// TwinCAT 3 PLC project Untitled1
// ProgramVersion: 3.1.4023.0
// libraries:
//   Tc2_MC2, * (Beckhoff Automation GmbH)
//   Tc2_Standard, * (Beckhoff Automation GmbH)
//   Tc2_System, * (Beckhoff Automation GmbH)
//   Tc2_Utilities, * (Beckhoff Automation GmbH)
//   Tc3_JsonXml, * (Beckhoff Automation GmbH)
//   Tc3_Module, * (Beckhoff Automation GmbH)
//   Tc3_PackML_V2, * (Beckhoff Automation GmbH)
// project tree:
//   DUTs/ Bundle.TcDUT (not stored), Interval.TcDUT (not stored), PositionMaterials.TcDUT (not stored)
//   DUTs/Enums/ TaskA22.TcDUT (not stored), Cardboard.TcDUT (not stored), CornerGuard.TcDUT (not stored), E_PMLCustomUnitMode.TcDUT (not stored), SectionEnum.TcDUT (not stored), Surface.TcDUT (not stored)
//   DUTs/Insertion Package/Drives/ AirPiston.TcPOU (not stored), ClearLinkMC.TcPOU (not stored), ServoNC.TcPOU (not stored), SimplePiston.TcPOU (not stored)
//   DUTs/Insertion Package/ Homing.TcDUT (not stored), Insertion.TcPOU (not stored), SuctionPad.TcDUT (not stored)
//   DUTs/Insertion Package/Prototypes/ FBA_Drive.TcPOU (not stored), FBA_TrifectaDrive.TcPOU (not stored), I_ContinuousDrive.TcIO (not stored), I_Drive.TcIO (not stored), I_EncodedDrive.TcIO (not stored), I_PositionalDrive.TcIO (not stored)
//   DUTs/Machines/ FoldingMachine.TcPOU, KukaRobot.TcPOU (not stored), RobotA22.TcPOU, WrapMachine.TcPOU
//   DUTs/Material Holders/ MaterialHolder.TcPOU (not stored), MaterialSlot.TcDUT (not stored), SkidMagazine.TcPOU (not stored)
//   GVLs/ ContainerArrays.TcGVL, GVL.TcGVL (not stored), Hardware.TcGVL, Misc.TcGVL (not stored)
//   / PlcTask.TcTTO (not stored)
//   POUs/A22 - Cardboard + Guard/AOIs/ AOI_LoadCornerCardboard.TcPOU (not stored), AOI_LoadCornerGuard.TcPOU, AOI_LoadFlatCardboard.TcPOU
//   POUs/A22 - Cardboard + Guard/ FiberboardEx.TcPOU
//   POUs/ FB_System.TcPOU (not stored), MAIN.TcPOU, BundleToJson.TcPOU (not stored)
//   POUs/Hardware Calls/ SuctionQualityPtr.TcPOU (not stored), SetSuctionsPtrArr.TcPOU (not stored), CallHardwareModules.TcPOU, SuctionQuality.TcPOU (not stored), SetSuctions.TcPOU (not stored), SetupHardware.TcPOU (not stored)
//   POUs/Materials/ GetMaterialLength.TcPOU (not stored), GetMaterialLengthFromCode.TcPOU (not stored), GetPairMasterLength.TcPOU (not stored), GetPositionMasterLength.TcPOU (not stored), MatchesMaterialType.TcPOU (not stored)
//   POUs/Utility/ CEILING.TcPOU (not stored), IntegerBitAccess.TcPOU (not stored), IntegerToBoolArray.TcPOU (not stored), WithinTolerance.TcPOU (not stored)
// real-time tasks:
//   TASK PlcTask: cycle T#10ms, priority 20, ADS port 350
// motion (NC):
//   TASK NC-Task 1 SAF: cycle T#2ms, priority 4, ADS port 501
//   TASK NC-Task 1 SVB: cycle T#10ms, priority 8, ADS port 511
//   AXIS A22_IM_HS_L (id 1)
//     OtherSettings: AllowMotionCmdToSlave=true
//     encoder EncType=19
//       EncPara: MaxCount=#xffffffff
//     drive DrvType=16
//       DrvPara: MaxCount=#xffffffff
//         Analog: TorqueSetpointScale=10, ScaleFactorActTorque=0.1
//         TimeComp: TaskDelayCycles=1
//     controller CtrType=1
//       CtrPara: PriorControlFactor=1
//         Observer: BandWidth=20
//   AXIS A22_IM_HS_R (id 2)
//     OtherSettings: AllowMotionCmdToSlave=true
//     encoder EncType=19
//       EncPara: MaxCount=#xffffffff
//     drive DrvType=16
//       DrvPara: MaxCount=#xffffffff, DriveControlDWord=#x00000100
//         Analog: TorqueSetpointScale=10, ScaleFactorActTorque=0.1
//         TimeComp: TaskDelayCycles=1
//     controller CtrType=1
//       CtrPara: PriorControlFactor=1
//         Observer: BandWidth=20
// I/O:
//   DEVICE Device 1 (EtherCAT) (disabled), AmsNetId 192.168.101.188.2.1
//     EK1200 [EK1200-5000 EtherCAT Power supply (2A E-Bus)]
//       IPC_O [EL2809 16Ch. Dig. Output 24V, 0.5A]
//       JUNC_1 [EK1122 2 port EtherCAT junction]
//         A21_C4 [EK1100 EtherCAT Coupler (2A E-Bus)]
//           A21_C4_I1 [EL1809 16Ch. Dig. Input 24V, 3ms]
//           A21_C4_O2 [EL2809 16Ch. Dig. Output 24V, 0.5A]
//           A21_C4_O3 [EL2809 16Ch. Dig. Output 24V, 0.5A]
//           BRIDGE_ROBOT1 [EL6695 EtherCAT Bridge terminal (Primary)]
//           A21_C4_END [EL9011 End Terminal]
//         A21_SB01 [EP1809-0021 16 Ch. Dig. Input 24V, 3ms, M8]
//         A21_SB05 [EP1008-0001 8 Ch. Dig. Input 24V, 3ms, M8]
//         A21_SB04 [EP1809-0021 16 Ch. Dig. Input 24V, 3ms, M8]
//         A21_SB03 [EP1008-0001 8 Ch. Dig. Input 24V, 3ms, M8]
//         A21_C1 [EK1100 EtherCAT Coupler (2A E-Bus)]
//           A21_C1_I1 [EL1809 16Ch. Dig. Input 24V, 3ms]
//           A21_C1_O2 [EL2809 16Ch. Dig. Output 24V, 0.5A]
//           BRIDGE_ROBOT2 [EL6695 EtherCAT Bridge terminal (Primary)]
//           A21_C1_END [EL9011 End Terminal]
//         A21_SB02 [EP1809-0021 16 Ch. Dig. Input 24V, 3ms, M8]
//         A21_SB07 [EP1008-0001 8 Ch. Dig. Input 24V, 3ms, M8]
//         A21_SB06 [EP1008-0001 8 Ch. Dig. Input 24V, 3ms, M8]
//       JUNC_2 [EK1122 2 port EtherCAT junction]
//         A22_C1 [EK1100 EtherCAT Coupler (2A E-Bus)]
//           A22_C1_I1 [EL1809 16Ch. Dig. Input 24V, 3ms]
//           A22_C1_O2 [EL2809 16Ch. Dig. Output 24V, 0.5A]
//           A22_C1_JUNC [EK1122 2 port EtherCAT junction]
//             A22_C4 [EK1100 EtherCAT Coupler (2A E-Bus)]
//               A22_C4_I1 [EL1809 16Ch. Dig. Input 24V, 3ms]
//               A22_C4_O2 [EL2809 16Ch. Dig. Output 24V, 0.5A]
//               A22_C4_O3 [EL2809 16Ch. Dig. Output 24V, 0.5A]
//               Term 31 (EL9011) [EL9011 End Terminal]
//             A22_C4_NC2 [CD02 EtherCAT Drive (CoE)]
//             A22_C4_NC1_TEMP [EK1100 EtherCAT Coupler (2A E-Bus)]
//               Term 34 (EL1008) [EL1008 8Ch. Dig. Input 24V, 3ms]
//               Term 35 (EL2008) [EL2008 8Ch. Dig. Output 24V, 0.5A]
//               Term 36 (EL9011) [EL9011 End Terminal]
//             A22_SB01 [EP1809-0021 16 Ch. Dig. Input 24V, 3ms, M8]
//             A22_SB04 [EP1809-0021 16 Ch. Dig. Input 24V, 3ms, M8]
//             A22_SB05 [EP1008-0001 8 Ch. Dig. Input 24V, 3ms, M8]
//             A22_C5 [EK1100 EtherCAT Coupler (2A E-Bus)]
//               A22_C5_I1 [EL1809 16Ch. Dig. Input 24V, 3ms]
//               A22_C5_O2 [EL2809 16Ch. Dig. Output 24V, 0.5A]
//               A22_C5_END [EL9011 End Terminal]
//             A22_SB06 [EP1008-0001 8 Ch. Dig. Input 24V, 3ms, M8]
//             A22_C6 [EK1100 EtherCAT Coupler (2A E-Bus)]
//               A22_C6_I1 [EL1809 16Ch. Dig. Input 24V, 3ms]
//               A22_C6_O2 [EL2809 16Ch. Dig. Output 24V, 0.5A]
//               A22_C6_O3 [EL2809 16Ch. Dig. Output 24V, 0.5A]
//               BRDIGE_ROBOT3 [EL6695 EtherCAT Bridge terminal (Primary)]
//               A22_C6_END [EL9011 End Terminal]
//             A22_SB08 [EP1008-0001 8 Ch. Dig. Input 24V, 3ms, M8]
//             A22_SB09 [EP2338-1001 8 Ch. Dig. Input/Output 24V, 3ms, 0,5A, M8]
//             A22_SB03 [EP1008-0001 8 Ch. Dig. Input 24V, 3ms, M8]
//             A22_SB02 [EP1809-0021 16 Ch. Dig. Input 24V, 3ms, M8]
//             A22_SB07 [EP1008-0001 8 Ch. Dig. Input 24V, 3ms, M8]
//             A22_C7 [EK1100 EtherCAT Coupler (2A E-Bus)]
//               A22_C7_I1 [EL1809 16Ch. Dig. Input 24V, 3ms]
//               A22_C7_O2 [EL2809 16Ch. Dig. Output 24V, 0.5A]
//               BRIDGE_ROBOT4 [EL6695 EtherCAT Bridge terminal (Primary)]
//               A22_C7_END [EL9011 End Terminal]
//   DEVICE Device 2 (TC3 EIP Scanner) (disabled), AmsNetId 192.168.101.188.3.1
//     ClearLink_A22 // <INFO> 169.254.0.152, ClearLink (ProdCode: 1, Rev: 2.93, Mac: 24:15:10:b0:30:37) </INFO> <EDS> C:\TwinCAT\3.1\Config\Io\EtherNetIP\clearlink_2.92.eds </EDS>
// variable links:
//   NC-Task 1 SAF/Axes/A22_IM_HS_R <-> Device 1 (EtherCAT)/EK1200/JUNC_2/A22_C1/A22_C1_JUNC/A22_C4_NC2
//     Drive/Inputs/In/nDataIn1 <-> TxPDO 1/Following Error Actual Value
//     Drive/Inputs/In/nDataIn3[0] <-> TxPDO 4/Torque Actual Value
//     Drive/Inputs/In/nDcOutputTime <-> InfoData/DcOutputShift
//     Drive/Inputs/In/nState1 <-> TxPDO 4/Statusword
//     Drive/Inputs/In/nState2 <-> TxPDO 4/Statusword @bit 8
//     Drive/Inputs/In/nState4 @bit 1 <-> WcState/InputToggle
//     Drive/Inputs/In/nState4 <-> WcState/WcState
//     Drive/Inputs/In/nState5 <-> TxPDO 3/Modes of Operation Display
//     Drive/Outputs/Out/nCtrl1 <-> RxPDO 4/Controlword
//     Drive/Outputs/Out/nCtrl2 <-> RxPDO 4/Controlword @bit 8
//     Drive/Outputs/Out/nCtrl5 <-> RxPDO 4/Modes of Operation
//     Drive/Outputs/Out/nDataOut1 <-> RxPDO 1/Target Position
//     Drive/Outputs/Out/nDataOut2 <-> RxPDO 2/Target Velocity
//     Drive/Outputs/Out/nDataOut3[0] <-> RxPDO 4/Torque Offset
//     Drive/Outputs/Out/nDataOut4[0] <-> RxPDO 3/Target Torque
//     Enc/Inputs/In/nDataIn1 <-> TxPDO 2/Position Actual Value
//     Enc/Inputs/In/nDcInputTime <-> InfoData/DcInputShift
//     Enc/Inputs/In/nState4 @bit 1 <-> WcState/InputToggle
//     Enc/Inputs/In/nState4 <-> WcState/WcState
//   Untitled1/Untitled1 Instance <-> Device 1 (EtherCAT)/EK1200/JUNC_2/A22_C1/A22_C1_JUNC/A22_C6/BRDIGE_ROBOT3
//     PlcTask Inputs/Hardware.robot3.inputs[{2..20}] <-> IO Inputs/In_{2..20}  (19 links)
//     PlcTask Inputs/Hardware.robot3.inputs[1] <-> IO Inputs/In
//     PlcTask Inputs/Hardware.robot3.offline <-> SYNC Inputs/External device not connected
//     PlcTask Outputs/Hardware.robot3.outputs[{2..20}] <-> IO Outputs/Out_{2..20}  (19 links)
//     PlcTask Outputs/Hardware.robot3.outputs[1] <-> IO Outputs/Out
//   Untitled1/Untitled1 Instance <-> Device 1 (EtherCAT)/EK1200/JUNC_2/A22_C1/A22_C1_JUNC/A22_C7/BRIDGE_ROBOT4
//     PlcTask Inputs/Hardware.robot4.inputs[{2..20}] <-> IO Inputs/In_{2..20}  (19 links)
//     PlcTask Inputs/Hardware.robot4.inputs[1] <-> IO Inputs/In
//     PlcTask Inputs/Hardware.robot4.offline <-> SYNC Inputs/External device not connected
//     PlcTask Outputs/Hardware.robot4.outputs[{2..20}] <-> IO Outputs/Out_{2..20}  (19 links)
//     PlcTask Outputs/Hardware.robot4.outputs[1] <-> IO Outputs/Out
//   Untitled1/Untitled1 Instance <-> Device 1 (EtherCAT)/EK1200/JUNC_2/A22_C1/A22_C1_JUNC/A22_SB01
//     PlcTask Inputs/Hardware.horizontalDriveA22Left.home <-> Channel 6/Input
//     PlcTask Inputs/Hardware.horizontalDriveA22Left.innerLimit <-> Channel 5/Input
//     PlcTask Inputs/Hardware.horizontalDriveA22Left.outerLimit <-> Channel 4/Input
//     PlcTask Inputs/Hardware.suctionA22BottomLeft[1].occupied <-> Channel 10/Input
//     PlcTask Inputs/Hardware.suctionA22BottomLeft[2].occupied <-> Channel 11/Input
//     PlcTask Inputs/Hardware.suctionA22BottomLeft[3].occupied <-> Channel 12/Input
//     PlcTask Inputs/Hardware.suctionA22TopLeft[1].occupied <-> Channel 7/Input
//     PlcTask Inputs/Hardware.suctionA22TopLeft[2].occupied <-> Channel 8/Input
//     PlcTask Inputs/Hardware.suctionA22TopLeft[3].occupied <-> Channel 9/Input
//     PlcTask Inputs/Hardware.verticalDriveA22Left.home <-> Channel 3/Input
//     PlcTask Inputs/Hardware.verticalDriveA22Left.innerLimit <-> Channel 2/Input
//     PlcTask Inputs/Hardware.verticalDriveA22Left.outerLimit <-> Channel 1/Input
//   Untitled1/Untitled1 Instance <-> Device 1 (EtherCAT)/EK1200/JUNC_2/A22_C1/A22_C1_JUNC/A22_SB02
//     PlcTask Inputs/Hardware.horizontalDriveA22Right.home <-> Channel 6/Input
//     PlcTask Inputs/Hardware.horizontalDriveA22Right.innerLimit <-> Channel 5/Input
//     PlcTask Inputs/Hardware.horizontalDriveA22Right.outerLimit <-> Channel 4/Input
//     PlcTask Inputs/Hardware.suctionA22BottomRight[1].occupied <-> Channel 10/Input
//     PlcTask Inputs/Hardware.suctionA22BottomRight[2].occupied <-> Channel 11/Input
//     PlcTask Inputs/Hardware.suctionA22BottomRight[3].occupied <-> Channel 12/Input
//     PlcTask Inputs/Hardware.suctionA22TopRight[1].occupied <-> Channel 7/Input
//     PlcTask Inputs/Hardware.suctionA22TopRight[2].occupied <-> Channel 8/Input
//     PlcTask Inputs/Hardware.suctionA22TopRight[3].occupied <-> Channel 9/Input
//     PlcTask Inputs/Hardware.verticalDriveA22Right.home <-> Channel 3/Input
//     PlcTask Inputs/Hardware.verticalDriveA22Right.innerLimit <-> Channel 2/Input
//     PlcTask Inputs/Hardware.verticalDriveA22Right.outerLimit <-> Channel 1/Input
//   Untitled1/Untitled1 Instance <-> Device 1 (EtherCAT)/EK1200/JUNC_2/A22_C1/A22_C1_JUNC/A22_SB06
//     PlcTask Inputs/Hardware.magazineA22Left.inPosition[1] <-> Channel 7/Input
//     PlcTask Inputs/Hardware.magazineA22Left.inPosition[2] <-> Channel 8/Input
//   Untitled1/Untitled1 Instance <-> Device 2 (TC3 EIP Scanner)/ClearLink_A22
//     PlcTask Inputs/Hardware.verticalDriveA22Left.hlfb <-> Connection 1 (Input/Output)/Inputs/Motor0 HLFB Duty
//     PlcTask Inputs/Hardware.verticalDriveA22Right.hlfb <-> Connection 1 (Input/Output)/Inputs/Motor1 HLFB Duty
//     PlcTask Outputs/Hardware.verticalDriveA22Left.outputRegister <-> Connection 1 (Input/Output)/Outputs/Motor0 Out Reg
//     PlcTask Outputs/Hardware.verticalDriveA22Left.pulse <-> Connection 1 (Input/Output)/Outputs/Motor0 Trig Pulses
//     PlcTask Outputs/Hardware.verticalDriveA22Right.outputRegister <-> Connection 1 (Input/Output)/Outputs/Motor1 Out Reg
//     PlcTask Outputs/Hardware.verticalDriveA22Right.pulse <-> Connection 1 (Input/Output)/Outputs/Motor1 Trig Pulses
//   Untitled1/Untitled1 Instance <-> NC-Task 1 SAF/Axes/A22_IM_HS_L
//     PlcTask Inputs/Hardware.horizontalDriveA22Left.axis.NcToPlc <-> Outputs/ToPlc
//     PlcTask Outputs/Hardware.horizontalDriveA22Left.axis.PlcToNc <-> Inputs/FromPlc
//   Untitled1/Untitled1 Instance <-> NC-Task 1 SAF/Axes/A22_IM_HS_R
//     PlcTask Inputs/Hardware.horizontalDriveA22Right.axis.NcToPlc <-> Outputs/ToPlc
//     PlcTask Outputs/Hardware.horizontalDriveA22Right.axis.PlcToNc <-> Inputs/FromPlc

// ---- GVLs/ContainerArrays.TcGVL
//{attribute 'qualified_only'}
VAR_GLOBAL //data arrays to be passed into material holder FBs - do not access directly
	skidHmiA22Left, skidHmiA22Right AT %M* : ARRAY[1...Cardboard.size-1] OF MaterialSlot;
	magazineHmiA22Left, magazineHmiA22Right AT %M* : ARRAY[1..CornerGuard.size-1] OF MaterialSlot;
END_VAR

// ---- GVLs/Hardware.TcGVL
//{attribute 'qualified_only'}
VAR_GLOBAL
	robot3 : RobotA22;
	robot4 : RobotA22;
	
	benderA22Left : FoldingMachine;
	
	skidA22Left : SkidMagazine;
	skidA22Right : SkidMagazine;
	magazineA22Left : SkidMagazine;
	magazineA22Right : SkidMagazine;
	
	wrapperA22 : WrapMachine;
	
	horizontalDriveA22Left, horizontalDriveA22Right : ServoNC := (
		limitSensorDefaultState := TRUE);
		
	verticalDriveA22Left, verticalDriveA22Right : ClearLinkMC := (
		limitSensorDefaultState := TRUE, 
		homingDirectionOut := TRUE, //outwards (up)
		minPosition := (26*5 * 25.4),
		displacementPerRotation := 5,
		unitsPerPulse := 800); //800 counts = 1 rotation
		
	insertionA22Left, insertionA22Right : Insertion;
		
	pistonA22Bottom : SimplePiston;
	
	(*
	each of these suction arrays are composed of 3 suction pads
	[1] - top/bottom
	[2] - corner
	[3] - side
	*)
	suctionA22TopLeft : ARRAY[1..3] OF SuctionPad;
	suctionA22TopRight : ARRAY[1..3] OF SuctionPad;
	suctionA22BottomLeft : ARRAY[1..3] OF SuctionPad; 
	suctionA22BottomRight : ARRAY[1..3] OF SuctionPad;
	
	//bottom piston suctions, may not exist
	suctionA22Bottom : ARRAY[1..2] OF SuctionPad;
END_VAR

// ---- DUTs/Machines/RobotA22.TcPOU
FUNCTION_BLOCK RobotA22 EXTENDS KukaRobot
VAR_OUTPUT //from outputs array
	taskID : TaskA22;
	param1 : INT;
	param2 : INT;
	Xmm : INT;
	Ymm : INT;
	Zmm : INT;
	angle : INT;
	foldPosition0 : INT;
	foldPosition1 : INT;
END_VAR
VAR_OUTPUT //from inputs array
	tool : SectionEnum := SectionEnum.CARDBOARD_CORNERGUARD;
	suspendedMaterial : STRING;
	
	completedTask : TaskA22;
	eoatDistance : INT;
	cardboardAvailability : INT;
	cornerGuardAvailability : INT;
	materialAtHoldingPosition : INT;
	//grp6
	//grp7
	
	wrapSafetyIn : BOOL;
	
END_VAR
VAR //HMI data
	reservationEnum : SectionEnum;
	hmiTask : STRING;
	hmiTool : STRING;
END_VAR

{warning disable C0195}
SUPER^();

outputs[1] := taskID;
outputs[2] := param1;
outputs[3] := param2;
outputs[4] := Xmm;
outputs[5] := Ymm;
outputs[6] := Zmm;
outputs[7] := angle;
outputs[8] := foldPosition0;
outputs[9] := foldPosition1;

refreshParameters();

reservationEnum := reservation;
IF reservationEnum = SectionEnum.NULL_SECTION THEN
	hmiReservation := 'N/A';
ELSE
	hmiReservation := TO_STRING(reservationEnum);
END_IF

hmiTask := TO_STRING(taskID);
hmiTool := TO_STRING(tool);

{attribute 'monitoring' := 'call'}
PROPERTY Busy : BOOL
GET
VAR
	//emptyOutput : ARRAY[1..50] OF INT;
END_VAR
//Busy stays TRUE until outputs are cleared AND completed task has elapsed
//Ready is always inverse of Busy
refreshParameters();

Busy := taskID <> 0 OR completedTask <> 0;
END_GET
END_PROPERTY

METHOD changeEOAT : BOOL
VAR_INPUT
	targetTool : SectionEnum;
END_VAR
//fill in IO here

changeEOAT := TRUE;
END_METHOD

METHOD clearCommand : BOOL
VAR_INPUT
END_VAR
SUPER^.clearCommand();

refreshParameters();
END_METHOD

{attribute 'monitoring' := 'call'}
PROPERTY Done : BOOL
GET
refreshParameters();

Done :=
	completedTask = taskID AND
	taskID <> 0 AND
	completedTask <> 0;
END_GET
END_PROPERTY

{attribute 'monitoring' := 'call'}
PROPERTY HoldMaterial : STRING
GET
HoldMaterial := suspendedMaterial;
END_GET
SET
suspendedMaterial := HoldMaterial;
END_SET
END_PROPERTY

{attribute 'monitoring' := 'call'}
PROPERTY Ready : BOOL
GET
refreshParameters();

Ready := taskID = 0 AND completedTask = 0;
END_GET
END_PROPERTY

METHOD PRIVATE refreshParameters : BOOL
VAR_INPUT
END_VAR
{warning disable C0196}
taskID := outputs[1];
param1 := outputs[2];
param2 := outputs[3];
Xmm := outputs[4];
Ymm := outputs[5];
Zmm := outputs[6];
angle := outputs[7];
foldPosition0 := outputs[8];
foldPosition1 := outputs[9];

completedTask := inputs[1];
(*
eoatDistance := inputs[2];
magazineAvailability := inputs[3];
chipboardSkidInPosition := inputs[4];
materialAtHoldingPosition := inputs[5];
//robotEOAT := inputs[6];

strapSafetyIn := inputs[4].15;
*)
END_METHOD

METHOD setGroup : BOOL
VAR_INPUT
	group : INT;
	value : INT;
END_VAR
SUPER^.setGroup(group := group, value := value);

refreshParameters();
END_METHOD

METHOD setParameters : BOOL
VAR_INPUT
	newTaskID : INT;
	newParam1 : INT;
	newParam2 : INT;
	newXmm : INT;
	newYmm : INT;
	newZmm : INT;
	newAngle : INT;
	newStagingOccupancy : INT;
	newInsertionSuctionStatus : INT;
	newMagazineStatus : INT; //unused
	newInspectionValue : INT;
END_VAR
super^.setGroup(group := 1, value := newTaskID);
super^.setGroup(group := 2, value := newParam1);
super^.setGroup(group := 3, value := newParam2);
super^.setGroup(group := 4, value := newXmm);
super^.setGroup(group := 5, value := newYmm);
super^.setGroup(group := 6, value := newZmm);
super^.setGroup(group := 7, value := newAngle);

newStagingOccupancy.15 := NOT wrapperA22.enable AND NOT wrapperA22.execute;
super^.setGroup(group := 8, value := newStagingOccupancy);

super^.setGroup(group := 9, value := newInsertionSuctionStatus);
super^.setGroup(group := 10, value := newMagazineStatus);
super^.setGroup(group := 11, value := newInspectionValue);

refreshParameters();
END_METHOD

END_FUNCTION_BLOCK

// ---- DUTs/Machines/FoldingMachine.TcPOU
FUNCTION_BLOCK FoldingMachine
VAR_INPUT
	//enable AT %Q* : BOOL;
	//reset AT %Q* : BOOL;
	foldingPositions AT %Q* : ARRAY[0..1] OF INT;
	
	lifterExtend AT %Q* : BOOL;
	lifterHalf AT %Q* : BOOL;
	lifterRetract AT %Q* : BOOL;
	
	benderExtend AT %Q* : BOOL;
	benderRetract AT %Q* : BOOL;
END_VAR
VAR_OUTPUT
	activeMaterial : STRING;
	
	lifterExtended AT %I* : BOOL;
	lifterIntermediate AT %I* : BOOL;
	lifterRetracted AT %I* : BOOL;
	
	benderExtended AT %I* : BOOL;
	benderRetracted AT %I* : BOOL;
	
	suction : SuctionPad;
	
	occupied AT %I* : BOOL;
	manifoldOk AT %I* : BOOL;
	
	//ready AT %I* : BOOL;
	//busy AT %I* : BOOL;
	//done AT %I* : BOOL;	
END_VAR

METHOD setFoldingPositions : BOOL
VAR_INPUT
	foldPos0, foldPos1 : INT;
END_VAR
foldingPositions[0] := foldPos0;
foldingPositions[1] := foldPos1;
END_METHOD

END_FUNCTION_BLOCK

// ---- DUTs/Machines/WrapMachine.TcPOU
FUNCTION_BLOCK WrapMachine
VAR_INPUT
	bEnable : BOOL;
END_VAR
VAR_OUTPUT
	error AT %I* : BOOL;
	ready AT %I* : BOOL;
	busy AT %I* : BOOL;
	done (*AT %I**) : BOOL;
	home AT %I* : BOOL;
	
	rotations AT %Q* : INT;
	execute AT %Q* : BOOL;
	enable AT %Q* : BOOL;
	reset AT %Q* : BOOL;
	
	timeout : BOOL;
	
	overheadTray : MaterialSlot;
END_VAR
VAR
	holdPost : TON;
	timeoutDelay : TON;
	resetDelay : TP;
	
	start : BOOL;
	step : (SETUP, RUN, WAIT);
END_VAR
VAR_STAT CONSTANT
	maxDelay : TIME := T#30S;
	pulseWidth : TIME := T#500MS;
END_VAR

holdPost(IN:= , PT:= pulseWidth, Q=> , ET=> );
timeoutDelay(IN:= (step > 0), PT:= maxDelay, Q=> timeout, ET=> );

resetDelay(IN:= error AND NOT resetDelay.Q , PT:= pulseWidth, Q=> , ET=> );
reset := resetDelay.Q AND (resetDelay.ET > resetDelay.PT/2);

IF timeoutDelay.Q THEN
	timeoutDelay.IN := FALSE;
	timeout := TRUE;
	busy := FALSE;
	step := SETUP;
END_IF

enable := bEnable AND robot3.wrapSafetyIn AND robot4.wrapSafetyIn;

CASE step OF
	SETUP:
		busy := FALSE;
		IF error THEN
			reset := NOT reset;
			enable := FALSE;//NOT enable;
			
		ELSE
			reset := FALSE;
			
			IF start THEN
				start := FALSE;
				step := RUN;
			END_IF
			
		END_IF
	
	RUN:
		execute := TRUE;
		IF execute AND NOT home THEN
			execute := FALSE;
			step := WAIT;
		END_IF
		
	WAIT:
		IF home THEN
			holdPost.IN := TRUE;
			enable := FALSE;
			execute := FALSE;
		END_IF
		
		IF holdPost.Q THEN
			holdPost.IN := FALSE;
			done := TRUE;
			step := 0;
		END_IF
		
END_CASE

METHOD clear : BOOL
VAR_INPUT
END_VAR
(*
reset should be continuously called until machine returns evidence that it is ready again
machine is expected to not respond to reset signals if it is already in an idle state
*)
enable := FALSE;
execute := FALSE;

IF error THEN
	reset := NOT reset;
	clear := NOT error;

ELSE
	reset := FALSE;
	clear := TRUE;
	
END_IF
END_METHOD

{attribute 'monitoring' := 'call'}
PROPERTY Overhead : STRING
GET
Overhead := overheadTray.material;
END_GET
SET
overheadTray.material := Overhead;
END_SET
END_PROPERTY

METHOD wrap : BOOL
VAR_INPUT
	reqRotations : INT;
END_VAR
IF ready AND NOT busy AND NOT error THEN
	rotations := reqRotations;
	busy := TRUE;
	start := TRUE;
	wrap := TRUE;
END_IF
END_METHOD

END_FUNCTION_BLOCK

// ---- POUs/A22 - Cardboard + Guard/AOIs/AOI_LoadCornerGuard.TcPOU
FUNCTION_BLOCK AOI_LoadCornerGuard
VAR_INPUT
	execute : BOOL;
END_VAR
VAR_IN_OUT CONSTANT
	sectionID : SectionEnum;
END_VAR
VAR_IN_OUT
	robot : RobotA22;
	magazine : SkidMagazine;
	loadedMaterials : ARRAY[*] OF STRING;
END_VAR
VAR_INPUT
	surfaceID : Surface;
	material : STRING;
	
	suctions : POINTER TO SuctionPad; //access from 0 to numPads-1, not LOWER_BOUND to UPPER_BOUND
	numPads : DINT;
END_VAR
VAR_OUTPUT
	donePulse : BOOL; //this signal turns on 1 cycle after done turns true, should not affect the program structure
	done : BOOL;
	busy : BOOL;
	error : BOOL;
	
	recovery : BOOL;
	failCounter : INT;
END_VAR
VAR
	run : BOOL;
	trigger : R_TRIG;
	doneTrigger : R_TRIG;
	
	column : INT;
	
	suctionTimer : TON;
	step : (IDLE, PREP_ROBOT, GET_FROM_STORAGE, LOAD_TO_INSERTION, COMPLETE, RECOVERY_IDLE, RECOVERY_REMOVE, RECOVERY_LOAD);
	
	i : DINT;
END_VAR
VAR CONSTANT
	suctionDelay : TIME := T#2S;
	suctionDistance : INT := 10;
END_VAR

{warning disable C0371}

trigger(CLK:= execute, Q=> );
doneTrigger(CLK:= done, Q=> donePulse);
busy := trigger.Q OR step > 0;

IF step > IDLE AND_THEN NOT preExecution() THEN //conditions to track before execution
	RETURN;
END_IF

(*
if required bunk was not found on table - restage entire table
if bunk was not loaded correctly - remove bunk, then restage entire table
*)
CASE step OF
	IDLE:
		IF trigger.Q THEN
			recovery := FALSE;
			done := FALSE;
			error := FALSE;
			step := PREP_ROBOT;
		END_IF
		
	PREP_ROBOT:
		robot.clearCommand();
		IF robot.Ready THEN
			step := GET_FROM_STORAGE;
			column := 0;
		END_IF
		
	GET_FROM_STORAGE:		
		IF NOT magazine.findSlot(material := material, index => column) THEN
			error := TRUE;
			RETURN;
		END_IF
		
		IF robot.eoatDistance < suctionDistance THEN //move from table to robot gripper
			robot.HoldMaterial := magazine.getSlot(i := column, error => );
		END_IF
		
		IF robot.Done THEN
			step := COMPLETE;
			RETURN;
		ELSIF robot.materialAtHoldingPosition > 0 THEN
			step := LOAD_TO_INSERTION;
			RETURN;
		END_IF
		
		CASE surfaceID OF
			Surface.TOP_LEFT, Surface.TOP_RIGHT:			robot.setGroup(group := 1, value := TaskA22.LOAD_CORNER_GUARD_UPPER);
			Surface.BOTTOM_LEFT, SURFACE.BOTTOM_RIGHT:		robot.setGroup(group := 1, value := TaskA22.LOAD_CORNER_GUARD_LOWER);
		END_CASE
		robot.setGroup(group := 2, value := column); 
			
	LOAD_TO_INSERTION:
		IF robot.materialAtHoldingPosition > 0 AND robot.HoldMaterial <> '' THEN //move from gripper to insertion
			loadedMaterials[surfaceID] := robot.HoldMaterial;
			robot.HoldMaterial := '';
		END_IF
		
		//numPads/3 <= i < numPads/3 * 2
		FOR i:=(numPads/3)*1 TO (numPads/3)*2-1 BY 1 DO //middle third suctions only
			suctions[i].enable := TRUE;
		END_FOR
		
		IF robot.Done THEN
			suctionTimer.IN := FALSE;
			step := COMPLETE;
			RETURN;
		END_IF
		
		suctionTimer(IN:= , PT:= suctionDelay, Q=> , ET=> );
		suctionTimer.IN := TRUE;
		
		IF suctionTimer.Q THEN
			robot.setGroup(group := 10, value := robot.materialAtHoldingPosition);
		END_IF
	
	COMPLETE:
		robot.clearCommand();
		
		IF //check insertion quality
			SuctionQualityPtr(
				suctions := suctions, 
				numPads := numPads, 
				insertionMaterial := loadedMaterials[surfaceID], 
				recipeMaterial := material)
		THEN
			done := TRUE;
			column := 0;
			step := 0;
			
		ELSE //recovery - remove and reload
			failCounter := failCounter + 1;
			step := RECOVERY_IDLE;
		END_IF
		
	//---------RECOVERY-----------------------------------------
	RECOVERY_IDLE:
		robot.clearCommand();
		IF robot.Ready THEN
			step := RECOVERY_REMOVE;
		END_IF
		
	RECOVERY_REMOVE:
		IF robot.Done THEN
			step := RECOVERY_LOAD;
			RETURN;
		END_IF
		
		CASE surfaceID OF
			Surface.TOP_LEFT, Surface.TOP_RIGHT:			robot.setGroup(group := 1, value := TaskA22.REMOVE_CORNER_GUARD_UPPER);
			Surface.BOTTOM_LEFT, SURFACE.BOTTOM_RIGHT:		robot.setGroup(group := 1, value := TaskA22.REMOVE_CORNER_GUARD_LOWER);
		END_CASE
		
	RECOVERY_LOAD:	
		recovery := TRUE;
		error := TRUE;
		
END_CASE

METHOD PRIVATE preExecution : BOOL
VAR_INPUT
END_VAR
{warning disable C0371}
IF material = '' THEN
	done := TRUE;
	RETURN;
END_IF

IF //robot must be ready before execution
	robot.error OR 
	robot.reservation <> sectionID OR 
	robot.tool <> sectionID
THEN
	error := TRUE;
	RETURN;
END_IF

preExecution := TRUE;
END_METHOD

METHOD reset : BOOL
VAR_INPUT
END_VAR
done := FALSE;
busy := FALSE;
error := FALSE;
recovery := FALSE;
failCounter := 0;

column := 0;
step := 0;
END_METHOD

END_FUNCTION_BLOCK

// ---- POUs/A22 - Cardboard + Guard/AOIs/AOI_LoadFlatCardboard.TcPOU
FUNCTION_BLOCK AOI_LoadFlatCardboard
VAR_INPUT
	execute : BOOL;
END_VAR
VAR_IN_OUT CONSTANT
	sectionID : SectionEnum;
END_VAR
VAR_IN_OUT
	robot : RobotA22;
	skid : SkidMagazine;
	loadedMaterials : ARRAY[*] OF STRING;
END_VAR
VAR_INPUT
	surfaceID : Surface;
	material : STRING;
	
	suctions : POINTER TO SuctionPad; //access from 0 to numPads-1, not LOWER_BOUND to UPPER_BOUND
	numPads : DINT;
END_VAR
VAR_OUTPUT
	donePulse : BOOL;
	done : BOOL;
	busy : BOOL;
	error : BOOL;
	
	recovery : BOOL;
	failCounter : INT;
END_VAR
VAR
	run : BOOL;
	trigger : R_TRIG;
	doneTrigger : R_TRIG;
	
	column : INT;
	
	suctionTimer : TON;
	step : (IDLE, PREP_ROBOT, GET_FROM_STORAGE, LOAD_TO_INSERTION, COMPLETE, RECOVERY_IDLE, RECOVERY_REMOVE, RECOVERY_WAIT, RECOVERY_LOAD);
	
	i : DINT;
END_VAR
VAR_STAT CONSTANT
	suctionDelay : TIME := T#2S;
	suctionDistance : INT := 10;
END_VAR

{warning disable C0371}

trigger(CLK:= execute, Q=> );
doneTrigger(CLK:= done, Q=> donePulse);
busy := trigger.Q OR step > 0;

IF step > IDLE AND_THEN NOT preExecution() THEN //conditions to track before execution
	RETURN;
END_IF

(*
if bunk was not loaded correctly - remove bunk, then restage entire table
*)
CASE step OF
	IDLE:
		IF trigger.Q THEN
			recovery := FALSE;
			done := FALSE;
			error := FALSE;
			step := PREP_ROBOT;
		END_IF
		
	PREP_ROBOT:
		robot.clearCommand();
		IF robot.Ready THEN
			step := GET_FROM_STORAGE;
			column := 0;
		END_IF
		
	GET_FROM_STORAGE:		
		IF NOT skid.findSlot(material := material, index => column) THEN
			error := TRUE;
			RETURN;
		END_IF
		
		IF robot.eoatDistance < suctionDistance THEN//move from table to robot gripper
			robot.HoldMaterial := skid.getSlot(i := column, error => );;
		END_IF
		
		IF robot.Done THEN
			step := COMPLETE;
			RETURN;
		ELSIF robot.materialAtHoldingPosition >= 1 AND robot.materialAtHoldingPosition <= 8 THEN
			step := LOAD_TO_INSERTION;
			RETURN;
		END_IF
		
		CASE surfaceID OF
			Surface.TOP_LEFT, Surface.TOP_RIGHT:			robot.setGroup(group := 1, value := TaskA22.LOAD_CORNER_GUARD_UPPER);
			Surface.BOTTOM_LEFT, SURFACE.BOTTOM_RIGHT:		robot.setGroup(group := 1, value := TaskA22.LOAD_CORNER_GUARD_LOWER);
		END_CASE
		robot.setGroup(group := 2, value := column); 
			
	LOAD_TO_INSERTION:
		IF robot.materialAtHoldingPosition > 0 AND robot.HoldMaterial <> '' THEN //move from gripper to insertion
			loadedMaterials[surfaceID] := robot.HoldMaterial;
			robot.HoldMaterial := '';
		END_IF
		
		//only bottom cardboard uses suction
		CASE surfaceID OF
			Surface.BOTTOM:		SetSuctionsPtrArr(suctions := suctions, numPads := numPads, state := TRUE);
		END_CASE
		
		IF robot.Done THEN
			suctionTimer.IN := FALSE;
			step := COMPLETE;
			RETURN;
		END_IF
		
		suctionTimer(IN:= , PT:= suctionDelay, Q=> , ET=> );
		suctionTimer.IN := TRUE;
		
		IF suctionTimer.Q THEN
			robot.setGroup(group := 10, value := robot.materialAtHoldingPosition);
		END_IF
	
	COMPLETE:
		robot.clearCommand();
		
		IF //if bottom then check insertion, otherwise done
			surfaceID <> Surface.BOTTOM OR_ELSE 
			SuctionQualityPtr(
				suctions := suctions, 
				numPads := numPads, 
				insertionMaterial := loadedMaterials[surfaceID], 
				recipeMaterial := material)
		THEN
			done := TRUE;
			column := 0;
			step := 0;
			
		ELSE //recovery - remove and reload
			failCounter := failCounter + 1;
			step := RECOVERY_IDLE;
		END_IF
		
	//---------RECOVERY-----------------------------------------
	RECOVERY_IDLE:
		robot.clearCommand();
		IF robot.Ready THEN
			step := RECOVERY_REMOVE;
		END_IF
		
	RECOVERY_REMOVE:
		IF robot.Done THEN
			step := RECOVERY_LOAD;
			RETURN;
		END_IF
		
		CASE surfaceID OF
			Surface.BOTTOM:		robot.setGroup(group := 1, value := TaskA22.REMOVE_CARDBOARD_BOTTOM);
		END_CASE
		
	RECOVERY_LOAD:	
		recovery := TRUE;
		error := TRUE;
		
END_CASE

METHOD PRIVATE preExecution : BOOL
VAR_INPUT
END_VAR
{warning disable C0371}
IF material = '' THEN
	done := TRUE;
	RETURN;
END_IF

IF //robot must be ready before execution
	robot.error OR 
	robot.reservation <> sectionID OR 
	robot.tool <> sectionID
THEN
	error := TRUE;
	RETURN;
END_IF

preExecution := TRUE;
END_METHOD

METHOD reset : BOOL
VAR_INPUT
END_VAR
done := FALSE;
busy := FALSE;
error := FALSE;
recovery := FALSE;
failCounter := 0;

column := 0;
step := 0;
END_METHOD

END_FUNCTION_BLOCK

// ---- POUs/A22 - Cardboard + Guard/FiberboardEx.TcPOU
FUNCTION_BLOCK FiberboardEx
VAR_IN_OUT
	benderLeft : FoldingMachine;
	
	robotLeft, robotRight : RobotA22;
	
	skidLeft, skidRight : SkidMagazine;
	magazineLeft, magazineRight : SkidMagazine;
	
	wrapper : WrapMachine;
	
	insertionLeft, insertionRight : Insertion;
	pistonBottom : SimplePiston;
	
	suctionTopLeft : ARRAY[*] OF SuctionPad; (*1..3*)
	suctionTopRight : ARRAY[*] OF SuctionPad; (*1..3*)
	suctionBottomLeft : ARRAY[*] OF SuctionPad; (*1..3*)
	suctionBottomRight : ARRAY[*] OF SuctionPad; (*1..3*)
	
	suctionBottom : ARRAY[*] OF SuctionPad; (*1..2*)
END_VAR
VAR_OUTPUT //controls
	pmlModeRequest : E_PMLCustomUnitMode := ePMLCustomUnitMode_Maintenance;
	pmlMode : E_PMLCustomUnitMode;
	
	pmlState : E_PMLState;
	pmlCommand : E_PMLCommand;

	stop : BOOL;
	execute : BOOL;
	hold : BOOL;
	reset : BOOL;
	
	done : BOOL;
	error : BOOL;
END_VAR
VAR
	pmlModeString : STRING;
	pmlStateString : STRING;
	
	pmlStateMachine : PML_StateMachine;
	pmlSemiAutoConfig : PML_UnitModeConfig;
	pmlModeManager : PML_UnitModeManager;
	
	step : (IDLE, LOAD_SIDES_CORNERS, LOAD_TOP_BOTTOM, PUSH, TARGET_WRAP_POSITION, WRAP_AND_RELEASE, COMPLETE := 1050);
	iPair : INT;
	
	masterLoadStep : INT;
	loadStepLeft, loadStepRight : INT;
	
	iWrap : INT;
	wrapPoints : INT;
	wrapRotations : INT;
	masterLength : INT;
	
	releaseDelayTimer : TON;
END_VAR
VAR //local types
	topLeftFoldsArr, topRightFoldsArr, bottomLeftFoldsArr, bottomRightFoldsArr : ARRAY[0..GVL.maxPairs] OF INT;
	materialsArr : ARRAY[0..GVL.maxPairs] OF PositionMaterials := [
		(
			position := 0,
			top := 'CAR20M',
			left := 'CAR20S',
			right := 'CAR20S',
			bottom := 'CAR20L',
			topLeft := 'CAR28M',
			topRight := 'CAR28S',
			bottomLeft := 'CAR28S',
			bottomRight := 'CAR28L',
			wrapPoints := 1,
			wrapRotations := 4
		),
		(
			position := 0,
			topLeft := 'COR48',
			topRight := 'COR48',
			bottomLeft := 'COR48',
			bottomRight := 'COR48'
		)];
	
	demoHeight : REAL := 640; //mm
	
	innerLoadedMaterials, outerLoadedMaterials : ARRAY[Surface.TOP..Surface.BOTTOM_RIGHT] OF STRING;
	//inner: cardboard by default
	//outer: corner guard by default
END_VAR
VAR CONSTANT
	sectionID : SectionEnum := SectionEnum.CARDBOARD_CORNERGUARD;
	releaseDelay : TIME := T#2000MS;
END_VAR
VAR
	//AOIs encapsulate functionality and reduce the number of module variables
	aoiCornerGuardLeft, aoiCornerGuardRight : AOI_LoadCornerGuard;
	aoiCornerCardboardLeft, aoiCornerCardboardRight : AOI_LoadCornerCardboard;
	aoiFlatCardboardLeft, aoiFlatCardboardRight : AOI_LoadFlatCardboard;
	
	//for testing only
	latchLeft, latchRight : BOOL; //prevents sliders from overshooting the inner limit sensor
	suctionEnableTopLeft, suctionEnableTopRight, suctionEnableBottomLeft, suctionEnableBottomRight : BOOL;
END_VAR

callLocalModules();

blocks();

configPML();
runPML();

ACTION blocks:
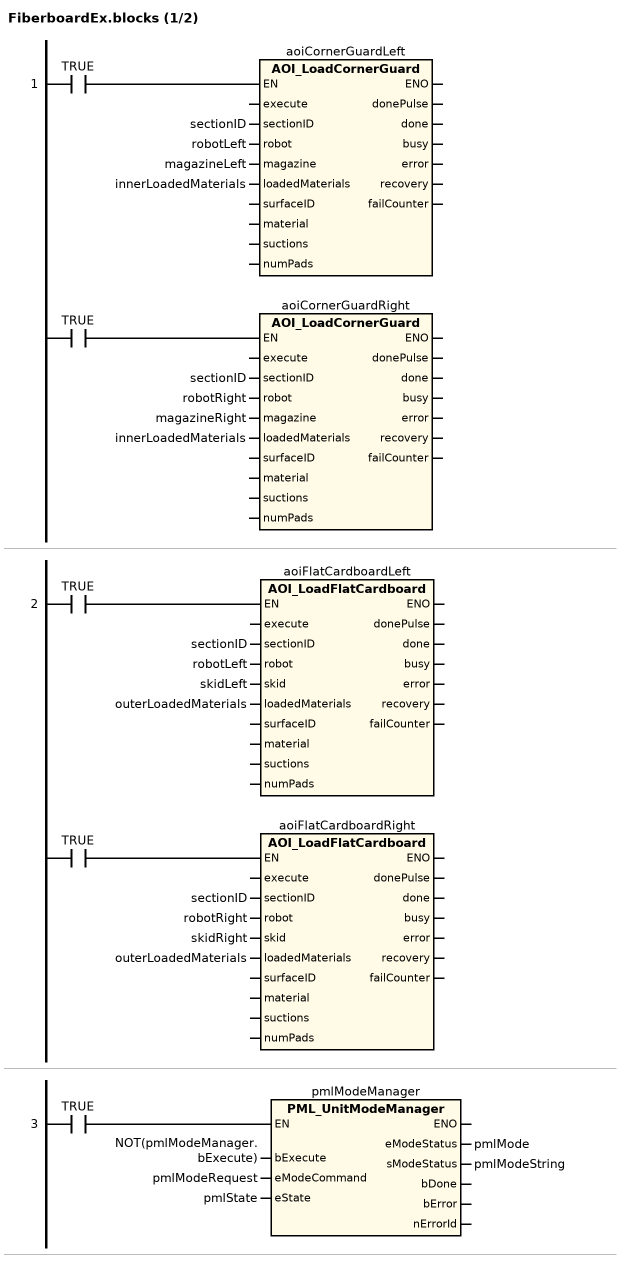
// NETWORK 1
aoiCornerGuardLeft(
    sectionID := sectionID,
    robot := robotLeft,
    magazine := magazineLeft,
    loadedMaterials := innerLoadedMaterials); // AOI_LoadCornerGuard
aoiCornerGuardRight(
    sectionID := sectionID,
    robot := robotRight,
    magazine := magazineRight,
    loadedMaterials := innerLoadedMaterials); // AOI_LoadCornerGuard

// NETWORK 2
aoiFlatCardboardLeft(
    sectionID := sectionID,
    robot := robotLeft,
    skid := skidLeft,
    loadedMaterials := outerLoadedMaterials); // AOI_LoadFlatCardboard
aoiFlatCardboardRight(
    sectionID := sectionID,
    robot := robotRight,
    skid := skidRight,
    loadedMaterials := outerLoadedMaterials); // AOI_LoadFlatCardboard

// NETWORK 3
pmlModeManager(
    bExecute := NOT(pmlModeManager.bExecute),
    eModeCommand := pmlModeRequest,
    eState := pmlState,
    eModeStatus => pmlMode,
    sModeStatus => pmlModeString); // PML_UnitModeManager

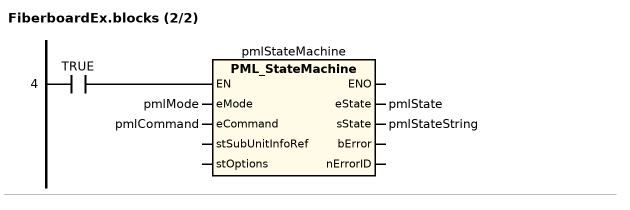
// NETWORK 4
pmlStateMachine(eMode := pmlMode, eCommand := pmlCommand, eState => pmlState, sState => pmlStateString); // PML_StateMachine
END_ACTION

ACTION callLocalModules:
{warning disable C0371}
END_ACTION

ACTION configPML:
pmlSemiAutoConfig(
	eMode:= 4, 
	sName:= 'SemiAuto', 
	bDisableClearing:= FALSE, 
	bDisableStarting:= FALSE, 
	bDisableSuspended:= FALSE, 
	bDisableStopping:= FALSE, 
	bDisableAborting:= FALSE, 
	bDisableHolding:= FALSE, 
	bDisableHeld:= FALSE, 
	bDisableUnholding:= FALSE, 
	bDisableSuspending:= FALSE, 
	bDisableUnsuspending:= FALSE, 
	bDisableResetting:= FALSE, 
	bDisableIdle:= FALSE, 
	bDisableCompleting:= FALSE, 
	bDisableComplete:= FALSE, 
	bEnableUnitModeChangeStopped:= TRUE, 
	bEnableUnitModeChangeIdle:= TRUE, 
	bEnableUnitModeChangeSuspended:= FALSE, 
	bEnableUnitModeChangeExecute:= FALSE, 
	bEnableUnitModeChangeAborted:= TRUE, 
	bEnableUnitModeChangeHeld:= FALSE, 
	bEnableUnitModeChangeComplete:= FALSE, 
	bError=> , 
	nErrorId=> );
END_ACTION

METHOD PROTECTED load : BOOL
VAR_INPUT
	pairIndex : INT;
END_VAR
VAR
	pair : REFERENCE TO PositionMaterials REF= materialsArr[pairIndex];
	nextPair : REFERENCE TO PositionMaterials;
END_VAR
(*
unlike other sections, the load() function for cardboard + corner guard only loads the corners
to load flat cardboards, use the function loadFlats()
*)
{warning disable C0371}

IF robotLeft.error OR robotRight.error THEN
	RETURN;
ELSIF NOT (robotLeft.reserve(sectionID) AND robotRight.reserve(sectionID)) THEN //both robots must be reserved first
	RETURN;
END_IF

IF pairIndex + 1 < GVL.maxPairs THEN
	nextPair REF= materialsArr[pairIndex + 1];
END_IF

CASE masterLoadStep OF
	0: //load this pair's side cardboards
		masterLoadStep := 10;
		IF
			loadFlatCardboardsEx(
				robot:= robotLeft, 
				aoiLoad:= aoiFlatCardboardLeft, 
				loadStep:= loadStepLeft, 
				pairIndex:= pairIndex, 
				includeTop:= FALSE, 
				includeLeft:= TRUE, 
				includeRight:= FALSE, 
				includeBottom:= FALSE, 
				error=> )
			AND
			loadFlatCardboardsEx(
				robot:= robotLeft, 
				aoiLoad:= aoiFlatCardboardLeft, 
				loadStep:= loadStepLeft, 
				pairIndex:= pairIndex, 
				includeTop:= FALSE, 
				includeLeft:= FALSE, 
				includeRight:= TRUE, 
				includeBottom:= FALSE, 
				error=> )
		THEN
			masterLoadStep := 10;
			loadStepLeft := loadStepRight := 0;
		END_IF
		
		
	10: //next pair (which is to be placed over this pair) has the same position as this pair
		IF pairIndex + 1 >= GVL.maxPairs THEN //no next pair - final pair is index 15 (16-1), not 16
			masterLoadStep := 20;
			loadStepLeft := loadStepRight := 0;
			
		ELSIF pair.position < nextPair.position THEN
			masterLoadStep := 20;
			loadStepLeft := loadStepRight := 0;
		(*	
		ELSIF MatchesMaterialType(pair:= nextPair, materialType:= 'CAR') AND_THEN loadCornerCardboards(pairIndex:= pairIndex + 1) THEN
			masterLoadStep := 20;
			loadStepLeft := loadStepRight := 0;
		*)
		ELSIF MatchesMaterialType(pair:= nextPair, materialType:= 'COR') AND_THEN loadCornerGuards(pairIndex:= pairIndex + 1) THEN
			masterLoadStep := 20;
			loadStepLeft := loadStepRight := 0;
			
		END_IF
		
	20: //load current pair
		IF
			MatchesMaterialType(pair:= pair, materialType:= 'CAR') AND_THEN loadCornerCardboards(pairIndex:= iPair) OR_ELSE
			MatchesMaterialType(pair:= pair, materialType:= 'COR') AND_THEN loadCornerGuards(pairIndex:= iPair)
		THEN //is cardboard
			loadStepLeft := loadStepRight := 0;
			masterLoadStep := COMPLETE;
		END_IF
	
	COMPLETE:
		robotLeft.release(sectionID);
		robotRight.release(sectionID);
		
		loadStepLeft := loadStepRight := 0;
		masterLoadStep := 0;
		load := TRUE;
	
END_CASE
END_METHOD

METHOD PROTECTED loadCornerCardboards : BOOL
VAR_INPUT
	pairIndex : INT;
END_VAR
VAR_OUTPUT
	error : BOOL;
END_VAR
VAR
	errorLeft, errorRight : BOOL;
	leftSuctionArr, rightSuctionArr : POINTER TO SuctionPad;
	leftNextSet, rightNextSet : INT;
	leftMaterial, rightMaterial : STRING;
	leftFold, rightFold : INT;
	
	pair : REFERENCE TO PositionMaterials REF= materialsArr[pairIndex];
	topLeftFold : INT := topLeftFoldsArr[pairIndex];
	topRightFold : INT := topRightFoldsArr[pairIndex];
	bottomLeftFold : INT := bottomLeftFoldsArr[pairIndex];
	bottomRightFold : INT := bottomRightFoldsArr[pairIndex];
END_VAR
{warning disable C0371}

loadCornerCardboards := 
	loadCornerCardboardsEx(
		robot:= robotLeft, 
		aoiLoad:= aoiCornerCardboardLeft, 
		loadStep:= loadStepLeft, 
		pairIndex:= pairIndex, 
		includeTopLeft:= TRUE, 
		includeTopRight:= FALSE, 
		includeBottomLeft:= TRUE, 
		includeBottomRight:= FALSE, 
		error=> errorLeft)
	AND
	loadCornerCardboardsEx(
		robot:= robotRight, 
		aoiLoad:= aoiCornerCardboardRight, 
		loadStep:= loadStepRight, 
		pairIndex:= pairIndex, 
		includeTopLeft:= FALSE, 
		includeTopRight:= TRUE, 
		includeBottomLeft:= FALSE, 
		includeBottomRight:= TRUE, 
		error=> errorLeft);
		
error := errorLeft OR errorRight;

(*
CASE cornerSetLeft OF
	0:
		leftNextSet := Surface.TOP_RIGHT;
		cornerSetLeft := 0;
		
	Surface.TOP_RIGHT: 
		leftNextSet := Surface.TOP_LEFT;
		leftSuctionArr := suctionTopRight;
		leftMaterial := pair.topRight;
		leftFold := topRightFold;
		
	Surface.TOP_LEFT: 
		leftNextSet := Surface.BOTTOM_RIGHT;
		leftSuctionArr := suctionTopLeft;
		leftMaterial := pair.topLeft;
		leftFold := topLeftFold;
		
	Surface.BOTTOM_RIGHT:
		leftNextSet := Surface.BOTTOM_LEFT;
		leftSuctionArr := suctionBottomRight;
		leftMaterial := pair.bottomRight;
		leftFold := bottomRightFold;
		
	Surface.BOTTOM_LEFT: 
		leftNextSet := COMPLETE;
		leftSuctionArr := suctionBottomLeft;
		leftMaterial := pair.bottomLeft;
		leftFold := bottomLeftFold;
END_CASE
IF
	(cornerSetLeft = 0 OR cornerSetLeft = COMPLETE) OR_ELSE
	leftCornerSequence(
		robot:= robotLeft, 
		skid:= skidLeft, 
		suctions := leftSuctionArr,
		loadStep:= loadStepLeft, 
		surfaceID:= cornerSetLeft,
		material:= pair.topRight, 
		foldPos0:= topRightFold, 
		foldPos1:= 0, 
		error=> )
THEN
	cornerSetLeft := leftNextSet;
	loadStepLeft := 0;
END_IF


CASE cornerSetRight OF
	0:
		cornerSetRight := Surface.TOP_RIGHT;
		rightSuctionArr := suctionTopRight;
		
	Surface.TOP_RIGHT:		
		rightNextSet := Surface.BOTTOM_RIGHT;
		rightSuctionArr := suctionTopRight;
		rightMaterial := pair.topRight;
		rightFold := topRightFold;
		
	Surface.BOTTOM_RIGHT: 
		rightNextSet := COMPLETE;
		rightSuctionArr := suctionBottomRight;
		rightMaterial := pair.bottomRight;
		rightFold := bottomRightFold;		
END_CASE
IF
	(cornerSetRight = 0 OR cornerSetRight = COMPLETE) OR_ELSE
	rightCornerSequence(
		robot:= robotRight, 
		skid:= skidRight, 
		suctions := rightSuctionArr,
		loadStep:= loadStepRight, 
		material:= pair.topRight, 
		surfaceID:= cornerSetRight,
		foldPos0:= pair.topRightFold, 
		foldPos1:= 0, 
		error=> )
THEN
	cornerSetRight := rightNextSet;
	loadStepRight := 0;
END_IF



IF cornerSetLeft = COMPLETE AND cornerSetRight = COMPLETE THEN
	loadCornerCardboards := TRUE;
	
	loadStepLeft := loadStepRight := 0;
	cornerSetLeft := cornerSetRight := 0;
END_IF
*)
END_METHOD

METHOD PROTECTED loadCornerCardboardsEx : BOOL
VAR_IN_OUT
	robot : RobotA22;
	aoiLoad : AOI_LoadCornerCardboard;
	loadStep : INT;
END_VAR
VAR_INPUT
	pairIndex : INT;
	includeTopLeft, includeTopRight, includeBottomLeft, includeBottomRight : BOOL;
END_VAR
VAR_OUTPUT
	error : BOOL;
END_VAR
VAR
	suctionsArrLeft, suctionsArrRight : POINTER TO SuctionPad;
	nextSetLeft, nextSetRight : INT;

	pair : REFERENCE TO PositionMaterials REF= materialsArr[pairIndex];
	topLeftFold : INT := topLeftFoldsArr[pairIndex];
	topRightFold : INT := topRightFoldsArr[pairIndex];
	bottomLeftFold : INT := bottomLeftFoldsArr[pairIndex];
	bottomRightFold : INT := bottomRightFoldsArr[pairIndex];
END_VAR
{warning disable C0371}

IF robot.error THEN
	error := TRUE;
	RETURN;
ELSIF robot.reservation <> sectionID AND_THEN NOT robot.reserve(sectionID) THEN
	RETURN;
ELSIF robot.tool <> sectionID AND_THEN NOT robot.changeEOAT(targetTool := sectionID) THEN
	RETURN;
END_IF

error := aoiLoad.error;

CASE loadStep OF
	0:
		loadStep := Surface.BOTTOM_LEFT;
		
	Surface.BOTTOM_LEFT:
		IF NOT includeBottomLeft OR aoiLoad.donePulse THEN
			aoiLoad.execute := FALSE;
			aoiLoad.material := '';
			loadStep := Surface.BOTTOM_RIGHT;
			RETURN;
		END_IF
		
		aoiLoad.surfaceID := loadStep;
		aoiLoad.material := pair.bottomLeft;
		aoiLoad.suctions := suctionBottomLeft;
		aoiLoad.numPads := UPPER_BOUND(suctionBottomLeft, 1) - LOWER_BOUND(suctionBottomLeft, 1) + 1;
		
		aoiLoad.foldPos0 := bottomLeftFold;
		aoiLoad.foldPos1 := 0;
		
		aoiLoad.execute := NOT aoiLoad.busy;
		
	Surface.BOTTOM_RIGHT:
		IF NOT includeBottomRight OR aoiLoad.donePulse THEN
			aoiLoad.execute := FALSE;
			aoiLoad.material := '';
			loadStep := Surface.TOP_LEFT;
			RETURN;
		END_IF
		
		aoiLoad.surfaceID := loadStep;
		aoiLoad.material := pair.bottomRight;
		aoiLoad.suctions := suctionBottomRight;
		aoiLoad.numPads := UPPER_BOUND(suctionBottomRight, 1) - LOWER_BOUND(suctionBottomRight, 1) + 1;
		
		aoiLoad.foldPos0 := bottomRightFold;
		aoiLoad.foldPos1 := 0;
		
		aoiLoad.execute := NOT aoiLoad.busy;
	
	Surface.TOP_LEFT:		
		IF NOT includeTopLeft OR aoiLoad.donePulse THEN
			aoiLoad.execute := FALSE;
			aoiLoad.material := '';
			loadStep := Surface.TOP_RIGHT;
			RETURN;
		END_IF
		
		aoiLoad.surfaceID := loadStep;
		aoiLoad.material := pair.top;
		aoiLoad.suctions := suctionTopLeft;
		aoiLoad.numPads := UPPER_BOUND(suctionTopLeft, 1) - LOWER_BOUND(suctionTopLeft, 1) + 1;
		
		aoiLoad.foldPos0 := topLeftFold;
		aoiLoad.foldPos1 := 0;
		
		aoiLoad.execute := NOT aoiLoad.busy;
		
	Surface.TOP_RIGHT:
		IF NOT includeTopRight OR aoiLoad.donePulse THEN
			aoiLoad.execute := FALSE;
			aoiLoad.material := '';
			loadStep := COMPLETE;
			RETURN;
		END_IF
		
		aoiLoad.surfaceID := loadStep;
		aoiLoad.material := pair.topRight;
		aoiLoad.suctions := suctionTopRight;
		aoiLoad.numPads := UPPER_BOUND(suctionTopRight, 1) - LOWER_BOUND(suctionTopRight, 1) + 1;
		
		aoiLoad.foldPos0 := topRightFold;
		aoiLoad.foldPos1 := 0;
		
		aoiLoad.execute := NOT aoiLoad.busy;
		
	COMPLETE:				
		robot.release(sectionID);
		
		aoiLoad.material := '';
		aoiLoad.execute := FALSE;
		
		loadCornerCardboardsEx := TRUE;
END_CASE
END_METHOD

METHOD loadCornerGuards : BOOL
VAR_INPUT
	pairIndex : INT;
END_VAR
VAR_OUTPUT
	error : BOOL;
END_VAR
VAR
	pair : REFERENCE TO PositionMaterials REF= materialsArr[pairIndex];
	errorLeft, errorRight : BOOL;
END_VAR
{warning disable C0371}

loadCornerGuards := 
	loadCornerGuardsEx(
		robot:= robotLeft, 
		aoiLoad:= aoiCornerGuardLeft, 
		loadStep:= loadStepLeft, 
		pairIndex:= pairIndex, 
		includeTopLeft:= TRUE, 
		includeTopRight:= FALSE, 
		includeBottomLeft:= TRUE, 
		includeBottomRight:= FALSE, 
		error=> errorLeft) 
	AND
	loadCornerGuardsEx(
		robot:= robotRight, 
		aoiLoad:= aoiCornerGuardRight, 
		loadStep:= loadStepRight, 
		pairIndex:= pairIndex, 
		includeTopLeft:= FALSE, 
		includeTopRight:= TRUE, 
		includeBottomLeft:= FALSE, 
		includeBottomRight:= TRUE, 
		error=> errorRight);
		
error := errorLeft OR errorRight;

(*
IF robotLeft.error OR robotRight.error THEN
	error := TRUE;
	RETURN;
	
ELSIF 
	(robotLeft.reservation <> sectionID AND_THEN NOT robotLeft.reserve(sectionID)) OR 
	(robotRight.reservation <> sectionID AND_THEN NOT robotRight.reserve(sectionID))
THEN //loading requires both robots be reserved together
	RETURN;
	
ELSIF //robots have wrong tool
	(robotLeft.tool <> sectionID AND_THEN NOT robotLeft.changeEOAT(targetTool := sectionID)) OR
	(robotRight.tool <> sectionID AND_THEN NOT robotRight.changeEOAT(targetTool := sectionID))
THEN
	RETURN;
	
END_IF

CASE loadStep OF
	0: //top and bottom
		IF aoiCornerGuardLeft.done AND aoiCornerGuardRight.done THEN
			aoiCornerGuardLeft.execute := aoiCornerGuardRight.execute := FALSE;
			aoiCornerGuardLeft.material := aoiCornerGuardRight.material := '';
			loadStep := 10;
			RETURN;
		END_IF
		
		aoiCornerGuardLeft.suctions := 0;
		aoiCornerGuardLeft.surfaceID := Surface.TOP;
		aoiCornerGuardLeft.material := pair.top;
		aoiCornerGuardLeft.numPads := 0;
		
		aoiCornerGuardRight.suctions := suctionBottom;
		aoiCornerGuardRight.surfaceID := Surface.BOTTOM;
		aoiCornerGuardRight.material := pair.bottom;
		aoiCornerGuardRight.numPads := 0;
		
		aoiCornerGuardLeft.execute := NOT aoiCornerGuardLeft.done AND NOT aoiCornerGuardLeft.busy;
		aoiCornerGuardRight.execute := NOT aoiCornerGuardRight.done AND NOT aoiCornerGuardRight.busy;
		
	10: //sides
		IF aoiCornerGuardLeft.done AND aoiCornerGuardRight.done THEN
			aoiCornerGuardLeft.execute := aoiCornerGuardRight.execute := FALSE;
			aoiCornerGuardLeft.material := aoiCornerGuardRight.material := '';
			loadStep := 10;
			RETURN;
		END_IF
		
		aoiCornerGuardLeft.suctions := 0;
		aoiCornerGuardLeft.surfaceID := Surface.LEFT;
		aoiCornerGuardLeft.material := pair.left;
		aoiCornerGuardLeft.numPads := 0;
		
		aoiCornerGuardRight.suctions := 0;
		aoiCornerGuardRight.surfaceID := Surface.RIGHT;
		aoiCornerGuardRight.material := pair.right;
		aoiCornerGuardRight.numPads := 0;
		
		aoiCornerGuardLeft.execute := NOT aoiCornerGuardLeft.done AND NOT aoiCornerGuardLeft.busy;
		aoiCornerGuardRight.execute := NOT aoiCornerGuardRight.done AND NOT aoiCornerGuardRight.busy;
		
	COMPLETE:
		loadStep := 0;
		loadCornerGuards := TRUE;
END_CASE

error := aoiCornerGuardLeft.error OR aoiCornerGuardRight.error;
*)
END_METHOD

METHOD loadCornerGuardsEx : BOOL
VAR_IN_OUT
	robot : RobotA22;
	aoiLoad : AOI_LoadCornerGuard;
	loadStep : INT;
END_VAR
VAR_INPUT
	pairIndex : INT;
	includeTopLeft, includeTopRight, includeBottomLeft, includeBottomRight : BOOL;
END_VAR
VAR_OUTPUT
	error : BOOL;
END_VAR
VAR
	pair : REFERENCE TO PositionMaterials REF= materialsArr[pairIndex];
END_VAR
{warning disable C0371}
IF robot.error THEN
	error := TRUE;
	RETURN;
ELSIF robot.reservation <> sectionID AND_THEN NOT robot.reserve(sectionID) THEN
	RETURN;
ELSIF robot.tool <> sectionID AND_THEN NOT robot.changeEOAT(targetTool := sectionID) THEN
	RETURN;
END_IF

error := aoiLoad.error;

CASE loadStep OF
	0:
		loadStep := Surface.BOTTOM_LEFT;
		
	Surface.BOTTOM_LEFT:
		IF NOT includeBottomLeft OR aoiLoad.donePulse THEN
			aoiLoad.execute := FALSE;
			aoiLoad.material := '';
			loadStep := Surface.BOTTOM_RIGHT;
			RETURN;
		END_IF
		
		aoiLoad.surfaceID := loadStep;
		aoiLoad.material := pair.bottomLeft;
		aoiLoad.suctions := suctionBottomLeft;
		aoiLoad.numPads := UPPER_BOUND(suctionBottomLeft, 1) - LOWER_BOUND(suctionBottomLeft, 1) + 1;
		
		aoiLoad.execute := NOT aoiLoad.busy;
		
	Surface.BOTTOM_RIGHT:
		IF NOT includeBottomRight OR aoiLoad.donePulse THEN
			aoiLoad.execute := FALSE;
			aoiLoad.material := '';
			loadStep := Surface.TOP_LEFT;
			RETURN;
		END_IF
		
		aoiLoad.surfaceID := loadStep;
		aoiLoad.material := pair.bottomRight;
		aoiLoad.suctions := suctionBottomRight;
		aoiLoad.numPads := UPPER_BOUND(suctionBottomRight, 1) - LOWER_BOUND(suctionBottomRight, 1) + 1;
		
		aoiLoad.execute := NOT aoiLoad.busy;
	
	Surface.TOP_LEFT:		
		IF NOT includeTopLeft OR aoiLoad.donePulse THEN
			aoiLoad.execute := FALSE;
			aoiLoad.material := '';
			loadStep := Surface.TOP_RIGHT;
			RETURN;
		END_IF
		
		aoiLoad.surfaceID := loadStep;
		aoiLoad.material := pair.top;
		aoiLoad.suctions := suctionTopLeft;
		aoiLoad.numPads := UPPER_BOUND(suctionTopLeft, 1) - LOWER_BOUND(suctionTopLeft, 1) + 1;
		
		aoiLoad.execute := NOT aoiLoad.busy;
		
	Surface.TOP_RIGHT:
		IF NOT includeTopRight OR aoiLoad.donePulse THEN
			aoiLoad.execute := FALSE;
			aoiLoad.material := '';
			loadStep := COMPLETE;
			RETURN;
		END_IF
		
		aoiLoad.surfaceID := loadStep;
		aoiLoad.material := pair.topRight;
		aoiLoad.suctions := suctionTopRight;
		aoiLoad.numPads := UPPER_BOUND(suctionTopRight, 1) - LOWER_BOUND(suctionTopRight, 1) + 1;
		
		aoiLoad.execute := NOT aoiLoad.busy;
		
	COMPLETE:				
		robot.release(sectionID);
		
		aoiLoad.material := '';
		aoiLoad.execute := FALSE;
		
		loadCornerGuardsEx := TRUE;
END_CASE
END_METHOD

METHOD PROTECTED loadFlatCardboards : BOOL
VAR_INPUT
	pairIndex : INT;
END_VAR
VAR_OUTPUT
	error : BOOL;
END_VAR
VAR
	pair : REFERENCE TO PositionMaterials REF= materialsArr[pairIndex];
	errorLeft, errorRight : BOOL;
END_VAR
{warning disable C0371}

loadFlatCardboards := 
	loadFlatCardboardsEx(
		robot:= robotLeft, 
		aoiLoad:= aoiFlatCardboardLeft, 
		loadStep:= loadStepLeft, 
		pairIndex:= pairIndex, 
		includeTop:= TRUE, 
		includeLeft:= FALSE, //left already loaded before
		includeRight:= FALSE, 
		includeBottom:= FALSE, 
		error=> errorLeft)
	AND
	loadFlatCardboardsEx(
		robot:= robotRight, 
		aoiLoad:= aoiFlatCardboardRight, 
		loadStep:= loadStepRight, 
		pairIndex:= pairIndex, 
		includeTop:= FALSE, 
		includeLeft:= FALSE, 
		includeRight:= FALSE, //right already loaded before
		includeBottom:= TRUE, 
		error=> errorRight);
		
error := errorLeft OR errorRight;

(*
IF robotLeft.error OR robotRight.error THEN
	error := TRUE;
	RETURN;
	
ELSIF 
	(robotLeft.reservation <> sectionID AND_THEN NOT robotLeft.reserve(sectionID)) OR 
	(robotRight.reservation <> sectionID AND_THEN NOT robotRight.reserve(sectionID))
THEN //loading requires both robots be reserved together
	RETURN;
	
ELSIF //robots have wrong tool
	(robotLeft.tool <> sectionID AND_THEN NOT robotLeft.changeEOAT(targetTool := sectionID)) OR
	(robotRight.tool <> sectionID AND_THEN NOT robotRight.changeEOAT(targetTool := sectionID))
THEN
	RETURN;
	
END_IF

CASE loadStep OF
	0: //top and bottom
		IF aoiFlatCardboardLeft.done AND aoiFlatCardboardRight.done THEN
			aoiFlatCardboardLeft.execute := aoiFlatCardboardRight.execute := FALSE;
			aoiFlatCardboardLeft.material := aoiFlatCardboardRight.material := '';
			loadStep := 10;
			RETURN;
		END_IF
		
		aoiFlatCardboardLeft.suctions := 0;
		aoiFlatCardboardLeft.surfaceID := Surface.TOP;
		aoiFlatCardboardLeft.material := pair.top;
		aoiFlatCardboardLeft.numPads := 0;
		
		aoiFlatCardboardRight.suctions := suctionBottom;
		aoiFlatCardboardRight.surfaceID := Surface.BOTTOM;
		aoiFlatCardboardRight.material := pair.bottom;
		aoiFlatCardboardRight.numPads := 0;
		
		aoiFlatCardboardLeft.execute := NOT aoiFlatCardboardLeft.done AND NOT aoiFlatCardboardLeft.busy;
		aoiFlatCardboardRight.execute := NOT aoiFlatCardboardRight.done AND NOT aoiFlatCardboardRight.busy;
		
	10: //sides
		IF aoiFlatCardboardLeft.done AND aoiFlatCardboardRight.done THEN
			aoiFlatCardboardLeft.execute := aoiFlatCardboardRight.execute := FALSE;
			aoiFlatCardboardLeft.material := aoiFlatCardboardRight.material := '';
			loadStep := 10;
			RETURN;
		END_IF
		
		aoiFlatCardboardLeft.suctions := 0;
		aoiFlatCardboardLeft.surfaceID := Surface.LEFT;
		aoiFlatCardboardLeft.material := pair.left;
		aoiFlatCardboardLeft.numPads := 0;
		
		aoiFlatCardboardRight.suctions := 0;
		aoiFlatCardboardRight.surfaceID := Surface.RIGHT;
		aoiFlatCardboardRight.material := pair.right;
		aoiFlatCardboardRight.numPads := 0;
		
		aoiFlatCardboardLeft.execute := NOT aoiFlatCardboardLeft.done AND NOT aoiFlatCardboardLeft.busy;
		aoiFlatCardboardRight.execute := NOT aoiFlatCardboardRight.done AND NOT aoiFlatCardboardRight.busy;
		
	COMPLETE:
		loadStepLeft := loadStepRight := 0;
		loadStep := 0;
		
		loadFlatCardboards := TRUE;
END_CASE

error := aoiFlatCardboardLeft.error OR aoiFlatCardboardRight.error;
*)
END_METHOD

METHOD loadFlatCardboardsEx : BOOL
VAR_IN_OUT
	robot : RobotA22;
	aoiLoad : AOI_LoadFlatCardboard;
	loadStep : INT;
END_VAR
VAR_INPUT
	pairIndex : INT;
	includeTop, includeLeft, includeRight, includeBottom : BOOL;
END_VAR
VAR_OUTPUT
	error : BOOL;
END_VAR
VAR
	pair : REFERENCE TO PositionMaterials REF= materialsArr[pairIndex];
END_VAR
IF robot.error THEN
	error := TRUE;
	RETURN;
ELSIF robot.reservation <> sectionID AND_THEN NOT robot.reserve(sectionID) THEN
	RETURN;
ELSIF robot.tool <> sectionID AND_THEN NOT robot.changeEOAT(targetTool := sectionID) THEN
	RETURN;
END_IF

error := aoiLoad.error;

CASE loadStep OF
	0:
		loadStep := Surface.TOP;
	
	Surface.TOP:	
		IF NOT includeTop OR aoiLoad.donePulse THEN
			aoiLoad.execute := FALSE;
			aoiLoad.material := '';
			loadStep := Surface.BOTTOM;
			RETURN;
		END_IF
		
		aoiLoad.surfaceID := Surface.TOP;
		aoiLoad.material := pair.top;
		aoiLoad.suctions := 0;
		aoiLoad.numPads := 0;
		
		aoiLoad.execute := NOT aoiLoad.busy;
		
	Surface.BOTTOM:
		IF NOT includeBottom OR aoiLoad.donePulse THEN
			aoiLoad.execute := FALSE;
			aoiLoad.material := '';
			loadStep := Surface.LEFT;
			RETURN;
		END_IF
		
		aoiLoad.surfaceID := Surface.BOTTOM;
		aoiLoad.material := pair.bottom;
		aoiLoad.suctions := suctionBottom;
		aoiLoad.numPads := UPPER_BOUND(suctionBottom, 1) - LOWER_BOUND(suctionBottom, 1) + 1;
		
		aoiLoad.execute := NOT aoiLoad.busy;
		
	Surface.LEFT:
		IF NOT includeLeft OR aoiLoad.donePulse THEN
			aoiLoad.execute := FALSE;
			aoiLoad.material := '';
			loadStep := Surface.RIGHT;
			RETURN;
		END_IF
		
		aoiLoad.surfaceID := Surface.LEFT;
		aoiLoad.material := pair.left;
		aoiLoad.suctions := 0;
		aoiLoad.numPads := 0;
		
		aoiLoad.execute := NOT aoiLoad.busy;
		
	Surface.RIGHT:
		IF NOT includeRight OR aoiLoad.donePulse THEN
			aoiLoad.execute := FALSE;
			aoiLoad.material := '';
			loadStep := COMPLETE;
			RETURN;
		END_IF
		
		aoiLoad.surfaceID := Surface.RIGHT;
		aoiLoad.material := pair.right;
		aoiLoad.suctions := 0;
		aoiLoad.numPads := 0;
		
		aoiLoad.execute := NOT aoiLoad.busy;
		
	COMPLETE:				
		robot.release(sectionID);
		
		aoiLoad.material := '';
		aoiLoad.execute := FALSE;
		
		loadFlatCardboardsEx := TRUE;
END_CASE
END_METHOD

METHOD PROTECTED maintenance : BOOL
VAR_INPUT
END_VAR
{warning disable C0371}
IF robotLeft.Done THEN
	robotLeft.clearCommand();
END_IF

IF robotRight.Done THEN
	robotRight.clearCommand();
END_IF
END_METHOD

METHOD manual : BOOL
VAR_INPUT
END_VAR
END_METHOD

METHOD PROTECTED process : BOOL
VAR_INPUT
	auto : BOOL;
END_VAR
VAR_OUTPUT
	error : BOOL;
END_VAR
{warning disable C0371}
(*
corrected sequence:
	load sides
	load corners
	load bottom
	load top
*)

CASE step OF
	IDLE:
		IF execute THEN
			execute := FALSE;
			step := LOAD_SIDES_CORNERS;
		END_IF
	
	LOAD_SIDES_CORNERS:
		IF
			(auto AND done) OR
			(NOT auto AND execute)
		THEN
			aoiCornerCardboardLeft.reset();
			aoiCornerCardboardRight.reset();
			
			aoiCornerGuardLeft.reset();
			aoiCornerGuardRight.reset();
			
			aoiFlatCardboardLeft.reset();
			aoiFlatCardboardRight.reset();
			
			step := LOAD_TOP_BOTTOM;
			RETURN;
		END_IF
		
		IF NOT done THEN
			done := load(pairIndex := iPair);
		END_IF
		
	LOAD_TOP_BOTTOM:
		IF
			(auto AND done) OR
			(NOT auto AND execute)
		THEN
			aoiCornerCardboardLeft.reset();
			aoiCornerCardboardRight.reset();
			
			aoiCornerGuardLeft.reset();
			aoiCornerGuardRight.reset();
			
			aoiFlatCardboardLeft.reset();
			aoiFlatCardboardRight.reset();
			
			step := PUSH;
			RETURN;
		END_IF
		
		IF NOT done THEN
			done := loadFlatCardboards(pairIndex := iPair);
		END_IF
		
	PUSH:
		IF
			(auto AND latchLeft AND latchRight AND pistonBottom.extended) OR
			(NOT auto AND execute)
		THEN
			step := TARGET_WRAP_POSITION;
			RETURN;
		END_IF
		
		insertionLeft.align(demoHeight+5);
		insertionRight.align(demoHeight+5);
		
		IF //align slider to 5mm gap above bundle height
			insertionLeft.sliderPos <> demoHeight+5 OR
			insertionRight.sliderPos <> demoHeight+5
		THEN
			RETURN;
		END_IF
		
		IF NOT latchLeft THEN
			latchLeft := insertionLeft.contact;
			insertionLeft.press();
		END_IF
		
		IF NOT latchRight THEN
			latchRight := insertionRight.contact;
			insertionRight.press();
		END_IF
		
		pistonBottom.extend();
		
	TARGET_WRAP_POSITION:		
		IF iWrap >= wrapPoints THEN
			step := COMPLETE;
			RETURN;
		END_IF
		
		//loadNextPair := materialsArr[iPair].position = materialsArr[iPair + 1].position;	
		
		IF materialsArr[iPair].position = materialsArr[iPair + 1].position THEN
			masterLength := MAX( GetPairMasterLength(materialsArr[iPair]), GetPairMasterLength(materialsArr[iPair + 1]) );
			wrapPoints := MAX( materialsArr[iPair].wrapPoints, materialsArr[iPair + 1].wrapPoints );
			wrapRotations := MAX( materialsArr[iPair].wrapRotations, materialsArr[iPair + 1].wrapRotations );
		ELSE
			masterLength := GetPairMasterLength(materialsArr[iPair]);
			wrapPoints := materialsArr[iPair].wrapPoints;
			wrapRotations := materialsArr[iPair].wrapRotations;
		END_IF
		
		(*
		directionCheckAndSet(
			wrapConveyorPos,
			(currentPair.position - masterLength/2) + (masterLength/(currentPair.wrapPoints + 1) * (iWrap + 1)));
		*)
		step := WRAP_AND_RELEASE;
		
	WRAP_AND_RELEASE:
		releaseDelayTimer(IN:= , PT:= releaseDelay, Q=> , ET=> );
		
		IF wrapper.ready THEN
			wrapper.wrap(wrapRotations);
			releaseDelayTimer.IN := TRUE;
		END_IF
		
		IF releaseDelayTimer.Q THEN
			SetSuctions(suctions := suctionTopLeft, state := FALSE);
			SetSuctions(suctions := suctionTopRight, state := FALSE);
			SetSuctions(suctions := suctionBottomLeft, state := FALSE);
			SetSuctions(suctions := suctionBottomRight, state := FALSE);
			
			insertionLeft.toHome();
			insertionRight.toHome();
			pistonBottom.retract();
		END_IF
		
		IF wrapper.done AND insertionLeft.home AND insertionRight.home AND pistonBottom.retracted THEN
			releaseDelayTimer.IN := FALSE;
			step := WRAP_AND_RELEASE;
		END_IF
	
	COMPLETE:
		iPair := (iPair + 1) MOD GVL.maxPairs;
		iWrap := wrapPoints := wrapRotations := 0;
		step := IDLE;
		
END_CASE
END_METHOD

METHOD PRIVATE ps_Aborting : BOOL
VAR_INPUT
END_VAR
{warning disable C0371}
insertionLeft.stop();
insertionRight.stop();
pistonBottom.stop();

aoiFlatCardboardLeft.reset();
aoiFlatCardboardRight.reset();

aoiCornerCardboardLeft.reset();
aoiCornerCardboardRight.reset();

aoiCornerGuardLeft.reset();
aoiCornerGuardRight.reset();

robotLeft.clearCommand();
robotRight.clearCommand();

//stop conveyors

ps_Aborting :=
	NOT insertionLeft.active AND
	NOT insertionRight.active AND
	NOT pistonBottom.busy AND
	NOT robotLeft.Busy AND
	NOT robotRight.Busy;
END_METHOD

METHOD PRIVATE ps_Clearing : BOOL
VAR_INPUT
END_VAR
{warning disable C0371}
insertionLeft.reset();
insertionRight.reset();

ps_Clearing := 
	NOT insertionLeft.error AND
	NOT insertionRight.error AND
	NOT wrapper.error AND
	NOT robotLeft.error AND
	NOT robotRight.error;
END_METHOD

METHOD PRIVATE ps_Execute : BOOL
VAR_INPUT
END_VAR
VAR_OUTPUT
	error : BOOL;
END_VAR
CASE pmlMode OF
	0: //invalid mode
	ePMLCustomUnitMode_Production:		ps_Execute := process(auto := TRUE, error => error);
	ePMLCustomUnitMode_Maintenance:		ps_Execute := maintenance();
	ePMLCustomUnitMode_Manual:			ps_Execute := manual();
	ePMLCustomUnitMode_SemiAuto:		ps_Execute := process(auto := FALSE, error => error);
END_CASE
END_METHOD

METHOD PRIVATE ps_Holding : BOOL
VAR_INPUT
END_VAR
{warning disable C0371}
insertionLeft.stop();
insertionRight.stop();
pistonBottom.stop();
//set robot to pause

ps_Holding :=
	NOT insertionLeft.active AND
	NOT insertionRight.active;
END_METHOD

METHOD PRIVATE ps_Resetting : BOOL
VAR_INPUT
END_VAR
{warning disable C0371}
insertionLeft.reset();
insertionRight.reset();

ps_Resetting := 
	reset AND
	NOT insertionLeft.error AND
	NOT insertionRight.error AND
	NOT wrapper.error AND
	NOT robotLeft.error AND
	NOT robotRight.error;
END_METHOD

METHOD PRIVATE ps_Starting : BOOL
VAR_INPUT
END_VAR
{warning disable C0371}
robotLeft.clearCommand();
robotRight.clearCommand();

insertionLeft.homingSequence();
insertionRight.homingSequence();
pistonBottom.retract();

ps_Starting := 
	insertionLeft.screw.HomeSet AND 
	insertionRight.screw.HomeSet AND 
	pistonBottom.retracted;
END_METHOD

METHOD PRIVATE ps_Stopping : BOOL
VAR_INPUT
END_VAR
{warning disable C0371}
insertionLeft.stop();
insertionRight.stop();
pistonBottom.stop();

aoiFlatCardboardLeft.reset();
aoiFlatCardboardRight.reset();

aoiCornerCardboardLeft.reset();
aoiCornerCardboardRight.reset();

aoiCornerGuardLeft.reset();
aoiCornerGuardRight.reset();

robotLeft.clearCommand();
robotRight.clearCommand();

wrapper.bEnable := FALSE;

//stop conveyors

ps_Stopping :=
	//NOT insertionLeft.active AND
	NOT insertionRight.active AND
	NOT pistonBottom.busy AND
	NOT robotLeft.Busy AND
	NOT robotRight.Busy AND
	NOT wrapper.busy;
END_METHOD

ACTION runPML:
(*
PackML
	state machine for packaging applications - see Tc3_PackML_V2 library on InfoSys
	
	final states - wait for an input or condition and command to new state
	intermediate states - complete a task and call pmlStateMachine.M_StateComplete() to advance to next state
	
the following states currently use the same logic (albeit in different methods), implementation may change later
	ps_Stopping() and ps_Aborting()
	ps_Resetting() and ps_Clearing()
	
STOP - controlled stop **with intent to shutdown or vacate for extended time** induced by operator/HMI - otherwise use HOLD
ABORT - emergency stop due to machine errors


HOLD - minor local issues
SUSPEND - external issues

EXECUTE - major control logic
	different modes may require different tasks
	create methods as required for different modes, then call the correct method in ps_Completing()
	can be commanded to STOP, ABORT, HOLD, or SUSPEND at any point
COMPLETING - process complete, move product out of system and finish transition to COMPLETED
*)

IF //abort at machine error
	//insertionLeft.error OR 
	insertionRight.error OR 
	robotLeft.error OR 
	robotRight.error OR
	wrapper.error
THEN
	pmlCommand := ePMLCommand_Abort;
	
ELSIF stop THEN //stop at command stop
	pmlCommand := ePMLCommand_Stop;

ELSIF FALSE (*A2.1 cannot allow bundles to enter*) THEN //FALSE condition never executes - this is temporary
	pmlCommand := ePMLCommand_Suspend;
END_IF


CASE pmlState OF
	0: (*ePMLState_Undefined*) //default state on startup
		pmlCommand := ePMLCommand_Stop;
		
	ePMLState_Stopping:
		IF ps_Stopping() THEN
			pmlStateMachine.M_StateComplete();
		END_IF
		
	ePMLState_Stopped:
		pmlCommand := ePMLCommand_Reset;
	
    ePMLState_Resetting:
		IF ps_Resetting() THEN
			reset := FALSE;
			pmlStateMachine.M_StateComplete();
		END_IF
		
	ePMLState_Idle:
		IF execute THEN
			execute := FALSE;
			pmlCommand := ePMLCommand_Start;
		END_IF		
	
	ePMLState_Starting:
		IF ps_Starting() THEN
			pmlStateMachine.M_StateComplete();
		END_IF
	
	ePMLState_Execute: 
		IF hold THEN
			pmlCommand := ePMLCommand_Hold;
		END_IF
		
		IF ps_Execute(error => error) THEN
			pmlStateMachine.M_StateComplete();
			pmlCommand := ePMLCommand_Complete;
		END_IF
		
	ePMLState_Completing:
		pmlStateMachine.M_StateComplete();
	
	ePMLState_Complete:
		pmlCommand := ePMLCommand_Reset;
	
	ePMLState_Holding:
		IF ps_Holding() THEN
			pmlStateMachine.M_StateComplete();
		END_IF
	
	ePMLState_Held:
		IF NOT hold THEN
			pmlCommand := ePMLCommand_Unhold;
		END_IF
	
	ePMLState_Unholding:
		pmlStateMachine.M_StateComplete(); //release all pause commands and IO
	
	ePMLState_Suspended: //based on output section conditions
	ePMLState_Suspending: //based on output section conditions
	ePMLState_Unsuspending: //based on output section conditions
	
	ePMLState_Aborting:
		IF ps_Aborting() THEN
			pmlStateMachine.M_StateComplete();
		END_IF
	
	ePMLState_Aborted:
		pmlCommand := ePMLCommand_Clear;
	
	ePMLState_Clearing:
		IF ps_Clearing() THEN
			pmlStateMachine.M_StateComplete();
		END_IF
	
END_CASE
END_ACTION

END_FUNCTION_BLOCK

// ---- POUs/MAIN.TcPOU
PROGRAM MAIN
VAR_OUTPUT
	currentTime : TIMESTRUCT;
END_VAR
VAR
	moduleA22 : FiberboardEx;
	
	getLocalTime : FB_LocalSystemTime;
END_VAR

CallHardwareModules(); //start program with hardware call

SetupHardware();

callModules();

CallHardwareModules(); //end program with hardware call

//BundleToJson();

ACTION callModules:
getLocalTime(
	sNetID:= '', 
	bEnable:= TRUE, 
	dwCycle:= , 
	dwOpt:= , 
	tTimeout:= , 
	bValid=> , 
	systemTime=> currentTime, 
	tzID=> );

moduleA22(
	benderLeft:= benderA22Left, 
	robotLeft:= robot3, 
	robotRight:= robot4, 
	skidLeft:= skidA22Left, 
	skidRight:= skidA22Right, 
	magazineLeft:= magazineA22Left, 
	magazineRight:= magazineA22Right, 
	wrapper:= wrapperA22, 
	insertionLeft:= insertionA22Left,
	insertionRight:= insertionA22Right,
	pistonBottom:= pistonA22Bottom, 
	suctionTopLeft:= suctionA22TopLeft, 
	suctionTopRight:= suctionA22TopRight, 
	suctionBottomLeft:= suctionA22BottomLeft, 
	suctionBottomRight:= suctionA22BottomRight, 
	suctionBottom:= suctionA22Bottom,
	pmlModeRequest=> , 
	pmlMode=> , 
	pmlState=> , 
	pmlCommand=> , 
	stop=> , 
	execute=> , 
	hold=> , 
	reset=> , 
	done=> , 
	error=> );
END_ACTION

END_PROGRAM

// ---- POUs/Hardware Calls/CallHardwareModules.TcPOU
FUNCTION CallHardwareModules : BOOL //only purpose of this function is to call modules from Hardware

robot3();
robot4();

skidA22Left(slots := skidHmiA22Left);
skidA22Right(slots := skidHmiA22Right);

magazineA22Left(slots := magazineHmiA22Left);
magazineA22Right(slots := magazineHmiA22Right);

wrapperA22();
benderA22Left();

verticalDriveA22Left();
verticalDriveA22Right();

horizontalDriveA22Left();
horizontalDriveA22Right();

pistonA22Bottom();

insertionA22Left(
	enable:= TRUE, 
	slider:= verticalDriveA22Left, 
	screw:= horizontalDriveA22Left, 
	contact=> , 
	active=> , 
	error=> , 
	home=> , 
	homingComplete=> , 
	sliderPos=> );
	
insertionA22Right(
	enable:= TRUE, 
	slider:= verticalDriveA22Right, 
	screw:= horizontalDriveA22Right, 
	contact=> , 
	active=> , 
	error=> , 
	home=> , 
	homingComplete=> , 
	sliderPos=> );

END_FUNCTION
